DATA_BLOCK "方向指示控制_DB"
{ S7_Optimized_Access := 'TRUE' }
VERSION : 0.1
NON_RETAIN
"方向指示控制"

BEGIN

END_DATA_BLOCK

